{attribute 'linkalways'} 
{attribute 'no_explicit_call' := 'This FB is a CLASS and must be accessed using methods or properties'}
FUNCTION_BLOCK PUBLIC Mc2Axis IMPLEMENTS Axis
VAR
	_axisRef : Tc2_MC2.Axis_Ref;
	_power : MC_Power;
	_jog : MC_Jog;
	_parameterSet : ST_AxisParameterSet;
	
	_enable : BOOL;
	_enablePositive : BOOL;
	_enableNegative : BOOL;
	
	_override : LREAL := 100.0;
	_bufferMode : AxisBufferMode := AxisBufferMode.Aborting;
	_powerBufferMode : MC_BufferMode := MC_Aborting;
	
	commandRunner : SingleAsyncCommandRunner;
END_VAR

PROPERTY PUBLIC _InternalAxisRef : REFERENCE TO Tc2_MC2.AXIS_REF
GET
_InternalAxisRef REF= _axisRef;
END_GET
END_PROPERTY

PROPERTY PUBLIC _InternalJog : REFERENCE TO MC_Jog
GET
_InternalJog REF= _jog;
END_GET
END_PROPERTY

PROPERTY PUBLIC _InternalParameterSet : REFERENCE TO ST_AxisParameterSet
GET
_InternalParameterSet REF= _parameterSet;
END_GET
END_PROPERTY

PROPERTY PUBLIC AreMotionCommandsLocked : BOOL
GET
AreMotionCommandsLocked := _axisRef.Status.MotionCommandsLocked;
END_GET
END_PROPERTY

PROPERTY AxisId : UDINT
GET
AxisId := _axisRef.NcToPlc.AxisId;
END_GET
END_PROPERTY

PROPERTY PUBLIC BufferMode : AxisBufferMode
GET // PUBLIC
BufferMode := _bufferMode;
END_GET
SET // PUBLIC
END_SET
END_PROPERTY

PROPERTY Busy : BOOL
GET
END_GET
END_PROPERTY

METHOD PUBLIC CyclicCall
VAR_INST
	_readParameterSet : MC_ReadParameterSet;
	parameterSetRead : BOOL;
END_VAR
THIS^._axisRef.ReadStatus();

THIS^._power(
	Axis := THIS^._axisRef,
	Enable := THIS^._enable,
	Enable_Positive := THIS^._enablePositive,
	Enable_Negative := THIS^._enableNegative,
	Override := THIS^._override,
	BufferMode := THIS^._powerBufferMode
);

IF NOT parameterSetRead THEN
	_readParameterSet(
		Axis := THIS^._axisRef,
		Parameter := _parameterSet,
		Execute := TRUE
	);
	
	IF NOT _readParameterSet.Busy THEN
		_readParameterSet(
			Axis := THIS^._axisRef,
			Parameter := _parameterSet,
			Execute := TRUE
		);
		IF _readParameterSet.Done THEN
			parameterSetRead := TRUE;
		END_IF
	END_IF
END_IF

commandRunner.CyclicCall();
END_METHOD

METHOD Disable
_enable := FALSE;
END_METHOD

METHOD DisableNegative
_enableNegative := FALSE;
END_METHOD

METHOD DisablePositive
_enablePositive := FALSE;
END_METHOD

METHOD Enable
VAR_INPUT
	bufferMode : AxisBufferMode;
END_VAR
_enable := TRUE;
_powerBufferMode := bufferMode;
END_METHOD

METHOD PUBLIC EnableNegative
_enableNegative := TRUE;
END_METHOD

METHOD EnablePositive
_enablePositive := TRUE;
END_METHOD

PROPERTY ErrorId : UDINT
GET
ErrorId := _axisRef.Status.ErrorID;
END_GET
END_PROPERTY

{warning 'add method implementation '}
METHOD PUBLIC Halt
END_METHOD

PROPERTY HasError : BOOL
GET
HasError := _axisRef.Status.Error;
END_GET
END_PROPERTY

METHOD HomingBuilder : I_HomingBuilder
VAR_INST
	builder : DefaultHomingBuilder(axis := THIS^);
END_VAR
HomingBuilder := builder;
END_METHOD

PROPERTY IsAccelerating : BOOL
GET
IsAccelerating := _axisRef.Status.Accelerating;
END_GET
END_PROPERTY

PROPERTY IsAtConstantVelocity : BOOL
GET
IsAtConstantVelocity := _axisRef.Status.ConstantVelocity;
END_GET
END_PROPERTY

PROPERTY IsAtStandStill : BOOL
GET
IsAtStandStill := _axisRef.Status.StandStill;
END_GET
END_PROPERTY

PROPERTY IsDecelerating : BOOL
GET
IsDecelerating := _axisRef.Status.Decelerating;
END_GET
END_PROPERTY

PROPERTY IsErrorStopped : BOOL
GET
IsErrorStopped := _axisRef.Status.ErrorStop;
END_GET
END_PROPERTY

PROPERTY IsHoming : BOOL
GET
IsHoming := _axisRef.Status.Homing;
END_GET
END_PROPERTY

PROPERTY IsInContinuousMotion : BOOL
GET
IsInContinuousMotion := _axisRef.Status.ContinuousMotion;
END_GET
END_PROPERTY

PROPERTY IsInDiscreteMotion : BOOL
GET
IsInDiscreteMotion := _axisRef.Status.DiscreteMotion;
END_GET
END_PROPERTY

PROPERTY IsInSynchronizedMotion : BOOL
GET
IsInSynchronizedMotion := _axisRef.Status.SynchronizedMotion;
END_GET
END_PROPERTY

PROPERTY PUBLIC IsMoving : BOOL
GET
IsMoving := _axisRef.Status.Moving;
END_GET
END_PROPERTY

PROPERTY PUBLIC IsNotMoving : BOOL
GET
IsNotMoving := _axisRef.Status.NotMoving;
END_GET
END_PROPERTY

PROPERTY IsReady : BOOL
GET
IsReady := _power.Status;
END_GET
END_PROPERTY

PROPERTY IsStopping : BOOL
GET
IsStopping := _axisRef.Status.Stopping;
END_GET
END_PROPERTY

METHOD JogBackwards
VAR_INPUT
	velocity : LREAL;
END_VAR
_jog(
	Axis := _axisRef,
	JogForward := FALSE,
	JogBackwards := TRUE,
	Mode := MC_JOGMODE_CONTINOUS,
	Velocity := velocity
);
END_METHOD

METHOD JogForward
VAR_INPUT
	velocity : LREAL;
END_VAR
_jog(
	Axis := _axisRef,
	JogForward := TRUE,
	JogBackwards := FALSE,
	Mode := MC_JOGMODE_CONTINOUS,
	Velocity := velocity
);
END_METHOD

METHOD MoveBuilder : I_MoveBuilder
VAR_INST
	builder : DefaultMoveBuilder(axis := THIS^);
END_VAR
MoveBuilder := builder;
END_METHOD

PROPERTY Override : LREAL
GET
Override := _override;
END_GET
SET
_override := Override;
END_SET
END_PROPERTY

PROPERTY PRIVATE PowerBufferMode : AxisBufferMode
SET // PRIVATE
CASE PowerBufferMode OF
	AxisBufferMode.Aborting:
		_powerBufferMode := MC_Aborting;
		
	AxisBufferMode.BlendingHigh:
		_powerBufferMode := MC_BlendingHigh;
	
	AxisBufferMode.BlendingLow:
		_powerBufferMode := MC_BlendingLow;
	
	AxisBufferMode.BlendingNext:
		_powerBufferMode := MC_BlendingNext;
	
	AxisBufferMode.BlendingPrevious:
		_powerBufferMode := MC_BlendingPrevious;
	
	AxisBufferMode.Buffered:
		_powerBufferMode := MC_Buffered;
ELSE
	_powerBufferMode := MC_Aborting;
END_CASE
END_SET
END_PROPERTY

{warning 'add method implementation '}
METHOD PUBLIC Reset
END_METHOD

PROPERTY State : AxisState
GET
IF _axisRef.Status.Disabled THEN
	State := AxisState.Disabled;
ELSIF _axisRef.Status.StandStill THEN
	State := AxisState.StandStill;
ELSIF _axisRef.Status.Homing THEN
	State := AxisState.Homing;
ELSIF _axisRef.Status.DiscreteMotion THEN
	State := AxisState.DiscreteMotion;
ELSIF _axisRef.Status.ContinuousMotion THEN
	State := AxisState.ContinuousMotion;
ELSIF _axisRef.Status.SynchronizedMotion THEN
	State := AxisState.SynchronisedMotion;
ELSIF _axisRef.Status.Stopping THEN
	State := AxisState.Stopping;
ELSIF _axisRef.Status.ErrorStop THEN
	State := AxisState.ErrorStop;
END_IF
END_GET
END_PROPERTY

{warning 'add method implementation '}
METHOD PUBLIC Stop
END_METHOD

METHOD StopJogging
_jog(
	Axis := _axisRef,
	JogForward := FALSE,
	JogBackwards := FALSE,
);
END_METHOD

END_FUNCTION_BLOCK

(* stored: Version 1.1.0.1, ProductVersion 3.1.4026.13
   POU Mc2Axis: Id {87dec7ab-2bb1-0d31-2938-1890a79b704e}, SpecialFunc None
   Folder Actions: Id {e1569167-2211-09ee-37b1-4c4339082715}
   Folder Builders: Id {d9bdc931-ea42-07ff-35a8-3438b480a9fc}
   Folder Cyclic: Id {65d85241-5ec7-061f-222a-51206cf70483}
   Folder Internal Properties: Id {6b0e8e04-77c1-0846-2f12-2cbaf9313d96}
   Folder Properties: Id {a05b4f4e-832a-0d7b-08f0-fcd60b2f3013}
   Property _InternalAxisRef: Id {b3bbeafc-9730-07c8-1499-224d56450eb9}
   Get Get: Id {89ccb65e-6803-0662-02de-0572acfe7b07}
   Property _InternalJog: Id {e6776bc9-6c2a-0958-2148-3909d21e12e8}
   Get Get: Id {4e0c3a92-f030-0e3c-1b37-ad02b1de4a2b}
   Property _InternalParameterSet: Id {0244552f-4842-0c79-2f0d-201f028ad021}
   Get Get: Id {543be191-e80e-02ce-1c64-f2d58cc92009}
   Property AreMotionCommandsLocked: Id {e068a7ec-23e8-0ecc-32ac-f973e5c7a7ac}
   Get Get: Id {01b07aa1-3b7a-0234-338e-b85086b7bb3d}
   Property AxisId: Id {c7651a46-71b9-038e-1c43-719416bd9313}
   Get Get: Id {08ce0879-0334-07a2-3e17-2d197a5cdee9}
   Property BufferMode: Id {b1f1f2ee-8671-0f38-1c84-0027a48dc79d}
   Get Get: Id {cc18705b-94c3-03c8-0b00-277fc60e5cc7}
   Set Set: Id {4f98bf38-da1e-03d1-0720-74bd8cee984d}
   Property Busy: Id {c4d003b0-13e6-0403-18c6-10814a47e5b1}
   Get Get: Id {8a95928c-66f9-065e-2c55-8badc2447c9b}
   Method CyclicCall: Id {af276999-925b-08bd-17bf-78ee3aa8ecf5}
   Method Disable: Id {dfd4c51c-e2a5-05b8-1af6-9e83988a982c}
   Method DisableNegative: Id {218b07b4-9eeb-0b96-2e59-23b0c37cdaf4}
   Method DisablePositive: Id {160fc863-e928-0447-1015-888d81b0da3e}
   Method Enable: Id {a5c3e8af-292a-0234-1365-c1ddeaa54005}
   Method EnableNegative: Id {56d72356-6be9-004a-21d6-4971af63f75d}
   Method EnablePositive: Id {7f5e4ae6-3fcd-0845-1d4f-a376b24f45d0}
   Property ErrorId: Id {4e974fd3-8d80-02ad-2984-1eaab9c44e9c}
   Get Get: Id {55bb3685-dcbc-0212-2320-19bfcd975526}
   Method Halt: Id {6e198554-7ed7-0df2-3397-a214af34e68a}
   Property HasError: Id {fa0b9369-19cb-09a8-2292-f0d3f60b2ec9}
   Get Get: Id {a2d3c493-e70c-0d5f-247b-0e5b1d3aa013}
   Method HomingBuilder: Id {aae47e8f-b398-0ee8-0823-c84c63cec8d4}
   Property IsAccelerating: Id {fbf04ea3-6007-01fd-29d0-fe161721b726}
   Get Get: Id {52f16271-e131-0a0a-01bc-3cd66e8d37be}
   Property IsAtConstantVelocity: Id {e764362a-6cbf-0c00-0c83-efd684712d35}
   Get Get: Id {dd55372b-331c-0667-0c94-101f7a8005ad}
   Property IsAtStandStill: Id {6c5d7679-3bfd-0390-1782-cb4036d1dd9a}
   Get Get: Id {f939a0c7-4536-0474-3f78-4e9d5e7415e8}
   Property IsDecelerating: Id {adcddba3-fe69-0a09-14a8-4a30295b8fcb}
   Get Get: Id {a6dad4c8-177e-0096-0095-179eba89a658}
   Property IsErrorStopped: Id {bb6d4909-6ebb-05a8-0001-42ff9461b984}
   Get Get: Id {f4555f7d-24e6-0b6d-2cbe-d801387f687a}
   Property IsHoming: Id {87dc129c-5a86-08d0-2441-d338c157c521}
   Get Get: Id {6523adcd-d89d-01d8-2be8-cf8477e67853}
   Property IsInContinuousMotion: Id {f6766b6f-bc43-08d1-3cda-75677c5df5d8}
   Get Get: Id {2fb5d8ea-58df-03fe-23d6-b3855f2ae260}
   Property IsInDiscreteMotion: Id {15a091c4-87ff-0fb7-27c2-0536e6ee65ed}
   Get Get: Id {9812fc92-57d0-05ae-161c-ed9c2c2b4bac}
   Property IsInSynchronizedMotion: Id {d97eba9f-86f0-05be-07ba-6bf02ccac385}
   Get Get: Id {6af207d3-2e98-0336-0821-1820cbbf865d}
   Property IsMoving: Id {a3a0c316-6f59-0969-204c-0c2440c99de6}
   Get Get: Id {b5f4a50f-7c1b-093e-3861-b47b3f6a8444}
   Property IsNotMoving: Id {24267b20-f85b-0e6e-3d6c-91c8cd63fc9b}
   Get Get: Id {c983ccf1-345f-0da5-26a8-cadbc46bf292}
   Property IsReady: Id {74f97be6-bc7d-03c6-1b8e-e21e84d38998}
   Get Get: Id {4a91b63d-db67-0588-3b46-776265da59c9}
   Property IsStopping: Id {7bd4141b-8486-0c17-0f4b-4db95efdab36}
   Get Get: Id {a4c81dc3-75b6-0811-1bdf-cec7cb0deb68}
   Method JogBackwards: Id {9620d646-aa48-03df-3385-f07a97d02bc4}
   Method JogForward: Id {3bb28509-f394-048c-2dce-52e7cffef153}
   Method MoveBuilder: Id {72c7d57d-0767-0a77-3dea-8c74f80b6ae2}
   Property Override: Id {2c5fc82b-4d8d-0dbb-140f-7b3e1127ec82}
   Get Get: Id {62921f3d-3cda-0500-00c1-192a453ca953}
   Set Set: Id {ea458627-da75-09b4-2b7f-8dbe8dc788c0}
   Property PowerBufferMode: Id {5157b215-7d0d-0e1f-121d-5f1686fc6d17}
   Set Set: Id {c538fb21-b0d8-0ea1-193a-07d319e487ee}
   Method Reset: Id {6604903b-7ce4-0da2-17fb-9cad8a6d23aa}
   Property State: Id {923d9d97-a258-013c-2820-c25f80ecf56a}
   Get Get: Id {7e1d908c-51c9-085e-1dfc-e72822a46246}
   Method Stop: Id {95654571-560d-01a6-37cf-8e57cae66fe8}
   Method StopJogging: Id {7d9bdd4e-6ddd-0c31-0aa6-83c81383dead} *)
